(* IEC 61131-3 sources: julia_exos_development/test/suite/template_generation/expected/StringAndArray_c-static_py/StringAndA_0, 2 files *)

(* ---- StringAndArray.st ---- *)
PROGRAM _INIT

END_PROGRAM

PROGRAM _CYCLIC

    //Auto connect:
    //StringAndArrayCyclic_0.Enable := ExComponentInfo_0.Operational; // Component has been deployed and started up successfully

    StringAndArrayCyclic_0(pStringAndArray := ADR(StringAndArray_0));

    ExComponentInfo_0(ExTargetLink := ADR(gTarget_0), ExComponentLink := ADR(gStringAndArray_0), Enable := TRUE);

    ExDatamodelInfo_0(ExTargetLink := ADR(gTarget_0), Enable := TRUE, InstanceName := 'StringAndArray_0');

END_PROGRAM

PROGRAM _EXIT

    StringAndArrayCyclic_0(Enable := FALSE);

END_PROGRAM

(* ---- StringAndArray.var ---- *)
VAR
    StringAndArray_0 : StringAndArray;
    StringAndArrayCyclic_0 : StringAndArrayCyclic;
    ExComponentInfo_0 : ExComponentInfo;
    ExDatamodelInfo_0 : ExDatamodelInfo;
END_VAR
